// Implicitly generated code : DO NOT EDIT
FUNCTION CheckDivLReal : LREAL
VAR_INPUT
	divisor:LREAL;
END_VAR

// Implicitly generated code : Only an Implementation suggestion
{noflow}
IF divisor = 0 THEN
	CheckDivLReal:=1;
	G_Diag.uiCheckDivReal:=G_Diag.uiCheckDivReal+1;
ELSE
	CheckDivLReal:=divisor;
END_IF;
{flow}

END_FUNCTION

(* stored: Version 1.1.0.1, ProductVersion 3.1.4024.4
   POU CheckDivLReal: Id {cd2f5ddd-2b3b-408d-9b93-d6b47e103165}, SpecialFunc CheckDivReal64 *)
